{attribute 'qualified_only'}
VAR_GLOBAL CONSTANT
	DESCRIPTION_LEN : USINT := 40;
	MESSAGE_LEN : UDINT := 255;
	TIMEOUT_LABEL : STRING(Param_Error.LABEL_LEN) := 'Feedback Timeout';
	TIMEOUT_PRIORITY : E_ErrorPriority := E_ErrorPriority.HIGH;
END_VAR

(* stored: Version 1.1.0.1, ProductVersion 3.1.4024.12
   GVL Param_Actuator: Id {96dd3f82-34ad-42db-b60f-e0ec9e701401} *)
